(* IEC 61131-3 sources: ICSQuartz/benchmarks/oscat_basic_findb_num/src, 1 file *)

(* ---- program.st ---- *)
PROGRAM PLC_PRG
VAR_INPUT
    in_str: STRING;
END_VAR

FINDB_NUM(in_str);

END_PROGRAM
